// TIA Portal V19 export
TYPE "C701_VAR_IF_VAT_TYPIC"
   STRUCT
      STO { ExternalAccessible := 'False'; ExternalVisible := 'False'; ExternalWritable := 'False'} : Struct   // Opsomming van alle storingen
         A001 : Bool;   // Alarm lage druk expansievat verwarming
         A002 : Bool;   // Fout drukmeting expansievat verwarming
         A003 : Bool;   // Alarm lage druk expansievat koeling
         A004 : Bool;   // Fout drukmeting expansievat koeling
      END_STRUCT;
   END_STRUCT;
END_TYPE
